SUBAPPLICATION Q_BackgroundColour_EnableOk_A (* Leitet aus 2 Bools (Kanal aktiviert + Hardware-QO) eine 3-Farben-VT-Hintergrundfarbe ab: Weiss=deaktiviert / Gruen=aktiviert+QO TRUE / Rot=aktiviert+QO FALSE (Stoerung). Generisch fuer jeden Kanal mit Enable-Schalter + Status-LED (PWM, PI, ...). *)
  (* Standard: 61499-2; Description: Copyright (c) 2026 Meisterschulen am Ostbahnhof This program and the accompanying materials are made available under the terms of the Eclipse Public License 2.0 which is available at https://www.eclipse.org/legal/epl-2.0/ SPDX-License-Identifier: EPL-2.0 *)
  (* Version 1.1, 2026-08-31, Franz Höpfinger, Meisterschulen am Ostbahnhof, Die reine 2-Bool-zu-1-von-3-Werten-Logik ist jetzt in MyLib::sys::Select_EnableOk ausgelagert (generisch, nicht auf Farben beschraenkt) - dieser Baustein instanziiert sie nur noch mit den 3 Farben als Parameter und haengt Q_BackgroundColour dran *)
  PACKAGE MyLib::sys;
  IMPORT isobus::UT::Q::const::colours::COLOR_GREEN;
  IMPORT isobus::UT::Q::const::colours::COLOR_RED;
  IMPORT isobus::UT::Q::const::colours::COLOR_WHITE;
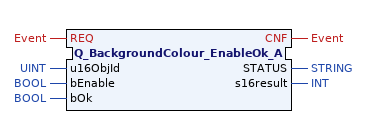
  EVENT_INPUT
    REQ; (* Neu auswerten - vom Aufrufer einmal pro moeglicher Aenderung von bEnable ODER bOk gefeuert (Schalter getoggelt, oder frisches QO eingetroffen), beide Werte werden zusammen mitgegeben *)
  END_EVENT
  EVENT_OUTPUT
    CNF; (* Farbe gesendet (Durchreichung von Q_BackgroundColour.CNF) *)
  END_EVENT
  VAR_INPUT
    u16ObjId : UINT; (* Object ID Status-Anzeige (CButton, nur Hintergrundfarbe, kein Text) - einmalig bei Instanziierung per Parameter gesetzt *)
    bEnable : BOOL; (* Kanal aktiviert (z.B. Enable-Flip-Flop.Q) *)
    bOk : BOOL; (* Hardware bestaetigt aktiv (z.B. logiBUS_..._IDA.QO) - nur relevant wenn bEnable=TRUE *)
  END_VAR
  VAR_OUTPUT
    STATUS : STRING; (* Service Status (Durchreichung von Q_BackgroundColour.STATUS) *)
    s16result : INT; (* Retval (Durchreichung von Q_BackgroundColour.s16result) *)
  END_VAR
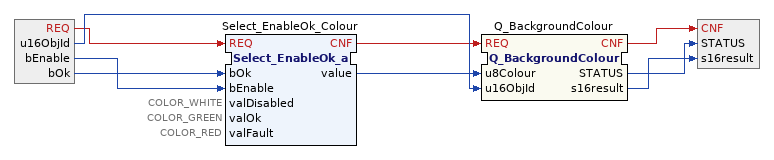
  FBS
    Q_BackgroundColour : isobus::UT::Q::Q_BackgroundColour;
  END_FBS
  SUBAPPS
    Select_EnableOk_Colour : MyLib::sys::Select_EnableOk_a(valDisabled := COLOR_WHITE, valOk := COLOR_GREEN, valFault := COLOR_RED);
  END_SUBAPPS
  EVENT_CONNECTIONS
    REQ TO Select_EnableOk_Colour.REQ;
    Select_EnableOk_Colour.CNF TO Q_BackgroundColour.REQ;
    Q_BackgroundColour.CNF TO CNF;
  END_CONNECTIONS
  DATA_CONNECTIONS
    bOk TO Select_EnableOk_Colour.bOk;
    bEnable TO Select_EnableOk_Colour.bEnable;
    Select_EnableOk_Colour.value TO Q_BackgroundColour.u8Colour;
    u16ObjId TO Q_BackgroundColour.u16ObjId;
    Q_BackgroundColour.STATUS TO STATUS;
    Q_BackgroundColour.s16result TO s16result;
  END_CONNECTIONS
END_SUBAPPLICATION
